// TIA Portal V16 export
// export: Created 2021-07-12T14:47:17.6242642Z, ExportSetting WithDefaults, DisplayName Totally Integrated Automation Portal, DisplayVersion V16, DisplayName TIA Portal Version Control Interface, DisplayVersion V16, DisplayName TIA Portal Openness, DisplayVersion V16, DisplayName STEP 7 Professional, DisplayVersion V16, DisplayName STEP 7 Safety, DisplayVersion V16, DisplayName WinCC Professional, DisplayVersion V16
VAR_GLOBAL   // PLC tag table "SimaHydTO_HydAxisServo_Interface"
   HydAxisServo_Actor_Interface_AddressIn AT %I1100.0 : "PD_TEL2_IN";   //    {ExternalWritable false}
   HydAxisServo_Sensor1_Interface_AddressIn AT %I1150.0 : "PD_TEL81_IN";   //    {ExternalWritable false}
   HydAxisServo_ForceSensor AT %IW1020 : Int;   //    {ExternalWritable false}
   HydAxisServo_Actor_Interface_AddressOut AT %Q1100.0 : "PD_TEL2_OUT";   //    {ExternalWritable false}
   HydAxisServo_Sensor1_Interface_AddressOut AT %Q1150.0 : "PD_TEL81_OUT";   //    {ExternalWritable false}
END_VAR
